REGION Network 61: Step[1301] : JOB[13] Condition
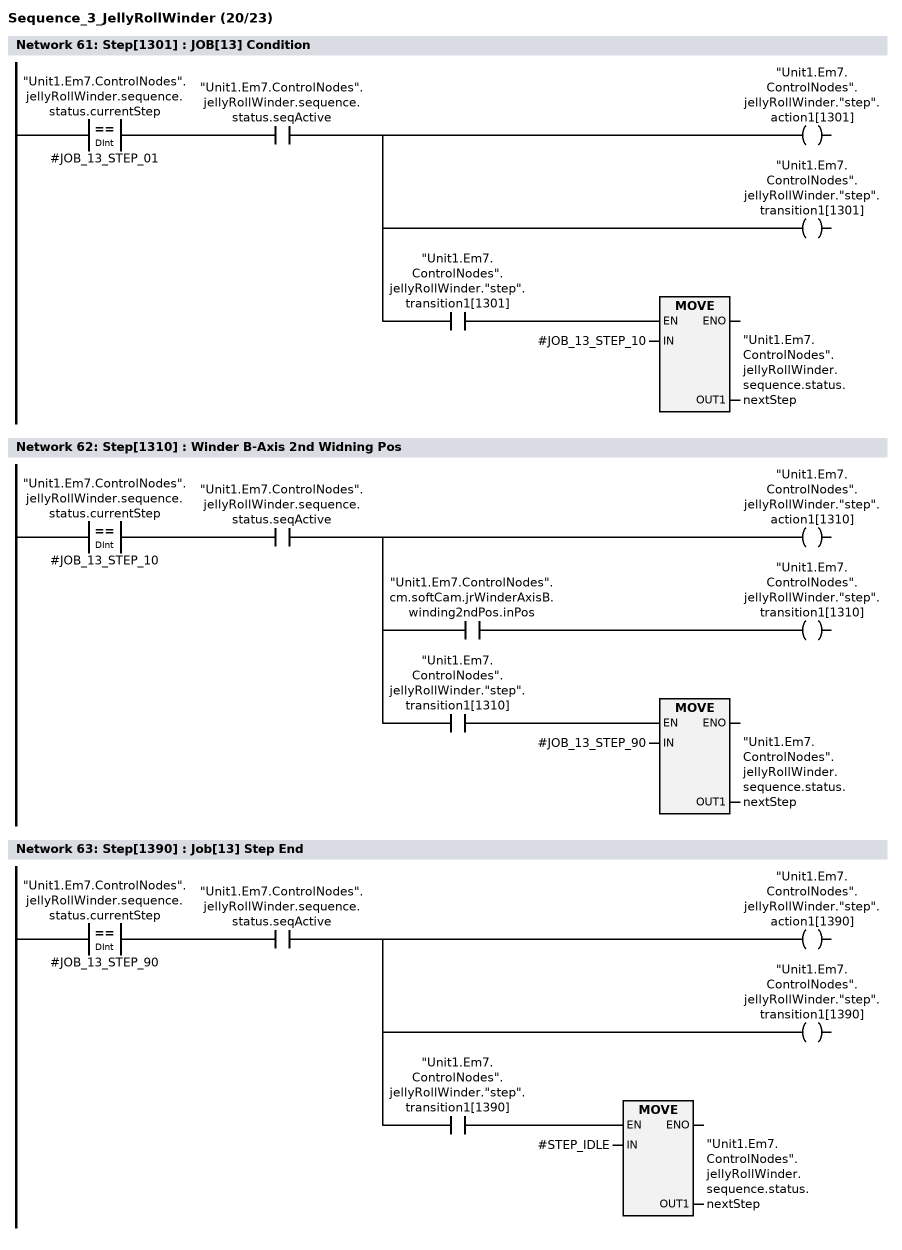
   RUNG wire#powerrail
      { S7_Templates := "SrcType := DInt" } EQ_Contact(in1 := "Unit1.Em7.ControlNodes".jellyRollWinder.sequence.status.currentStep, in2 := #JOB_13_STEP_01)
      Contact( "Unit1.Em7.ControlNodes".jellyRollWinder.sequence.status.seqActive )
      wire#w1
      Coil( "Unit1.Em7.ControlNodes".jellyRollWinder."step".action1[1301] )
   END_RUNG
   RUNG wire#w1
      Coil( "Unit1.Em7.ControlNodes".jellyRollWinder."step".transition1[1301] )
   END_RUNG
   RUNG wire#w1
      Contact( "Unit1.Em7.ControlNodes".jellyRollWinder."step".transition1[1301] )
      Move(in := #JOB_13_STEP_10, out1 => "Unit1.Em7.ControlNodes".jellyRollWinder.sequence.status.nextStep)
   END_RUNG
   // the same network as SCL:
   "Unit1.Em7.ControlNodes".jellyRollWinder."step".action1[1301] := ("Unit1.Em7.ControlNodes".jellyRollWinder.sequence.status.currentStep = #JOB_13_STEP_01) AND "Unit1.Em7.ControlNodes".jellyRollWinder.sequence.status.seqActive;
   "Unit1.Em7.ControlNodes".jellyRollWinder."step".transition1[1301] := ("Unit1.Em7.ControlNodes".jellyRollWinder.sequence.status.currentStep = #JOB_13_STEP_01) AND "Unit1.Em7.ControlNodes".jellyRollWinder.sequence.status.seqActive;
   IF ("Unit1.Em7.ControlNodes".jellyRollWinder.sequence.status.currentStep = #JOB_13_STEP_01) AND "Unit1.Em7.ControlNodes".jellyRollWinder.sequence.status.seqActive AND "Unit1.Em7.ControlNodes".jellyRollWinder."step".transition1[1301] THEN
       "Unit1.Em7.ControlNodes".jellyRollWinder.sequence.status.nextStep := #JOB_13_STEP_10;
   END_IF;
END_REGION

REGION Network 62: Step[1310] : Winder B-Axis 2nd Widning Pos
   RUNG wire#powerrail
      { S7_Templates := "SrcType := DInt" } EQ_Contact(in1 := "Unit1.Em7.ControlNodes".jellyRollWinder.sequence.status.currentStep, in2 := #JOB_13_STEP_10)
      Contact( "Unit1.Em7.ControlNodes".jellyRollWinder.sequence.status.seqActive )
      wire#w1
      Coil( "Unit1.Em7.ControlNodes".jellyRollWinder."step".action1[1310] )
   END_RUNG
   RUNG wire#w1
      Contact( "Unit1.Em7.ControlNodes".cm.softCam.jrWinderAxisB.winding2ndPos.inPos )
      Coil( "Unit1.Em7.ControlNodes".jellyRollWinder."step".transition1[1310] )
   END_RUNG
   RUNG wire#w1
      Contact( "Unit1.Em7.ControlNodes".jellyRollWinder."step".transition1[1310] )
      Move(in := #JOB_13_STEP_90, out1 => "Unit1.Em7.ControlNodes".jellyRollWinder.sequence.status.nextStep)
   END_RUNG
   // the same network as SCL:
   "Unit1.Em7.ControlNodes".jellyRollWinder."step".action1[1310] := ("Unit1.Em7.ControlNodes".jellyRollWinder.sequence.status.currentStep = #JOB_13_STEP_10) AND "Unit1.Em7.ControlNodes".jellyRollWinder.sequence.status.seqActive;
   "Unit1.Em7.ControlNodes".jellyRollWinder."step".transition1[1310] := ("Unit1.Em7.ControlNodes".jellyRollWinder.sequence.status.currentStep = #JOB_13_STEP_10) AND "Unit1.Em7.ControlNodes".jellyRollWinder.sequence.status.seqActive AND "Unit1.Em7.ControlNodes".cm.softCam.jrWinderAxisB.winding2ndPos.inPos;
   IF ("Unit1.Em7.ControlNodes".jellyRollWinder.sequence.status.currentStep = #JOB_13_STEP_10) AND "Unit1.Em7.ControlNodes".jellyRollWinder.sequence.status.seqActive AND "Unit1.Em7.ControlNodes".jellyRollWinder."step".transition1[1310] THEN
       "Unit1.Em7.ControlNodes".jellyRollWinder.sequence.status.nextStep := #JOB_13_STEP_90;
   END_IF;
END_REGION

REGION Network 63: Step[1390] : Job[13] Step End
   RUNG wire#powerrail
      { S7_Templates := "SrcType := DInt" } EQ_Contact(in1 := "Unit1.Em7.ControlNodes".jellyRollWinder.sequence.status.currentStep, in2 := #JOB_13_STEP_90)
      Contact( "Unit1.Em7.ControlNodes".jellyRollWinder.sequence.status.seqActive )
      wire#w1
      Coil( "Unit1.Em7.ControlNodes".jellyRollWinder."step".action1[1390] )
   END_RUNG
   RUNG wire#w1
      Coil( "Unit1.Em7.ControlNodes".jellyRollWinder."step".transition1[1390] )
   END_RUNG
   RUNG wire#w1
      Contact( "Unit1.Em7.ControlNodes".jellyRollWinder."step".transition1[1390] )
      Move(in := #STEP_IDLE, out1 => "Unit1.Em7.ControlNodes".jellyRollWinder.sequence.status.nextStep)
   END_RUNG
   // the same network as SCL:
   "Unit1.Em7.ControlNodes".jellyRollWinder."step".action1[1390] := ("Unit1.Em7.ControlNodes".jellyRollWinder.sequence.status.currentStep = #JOB_13_STEP_90) AND "Unit1.Em7.ControlNodes".jellyRollWinder.sequence.status.seqActive;
   "Unit1.Em7.ControlNodes".jellyRollWinder."step".transition1[1390] := ("Unit1.Em7.ControlNodes".jellyRollWinder.sequence.status.currentStep = #JOB_13_STEP_90) AND "Unit1.Em7.ControlNodes".jellyRollWinder.sequence.status.seqActive;
   IF ("Unit1.Em7.ControlNodes".jellyRollWinder.sequence.status.currentStep = #JOB_13_STEP_90) AND "Unit1.Em7.ControlNodes".jellyRollWinder.sequence.status.seqActive AND "Unit1.Em7.ControlNodes".jellyRollWinder."step".transition1[1390] THEN
       "Unit1.Em7.ControlNodes".jellyRollWinder.sequence.status.nextStep := #STEP_IDLE;
   END_IF;
END_REGION

REGION Network 64: *************** JOB[14] Cam Stop Sync ************************
END_REGION

REGION Network 65: Step[1401] : JOB[14] Condition
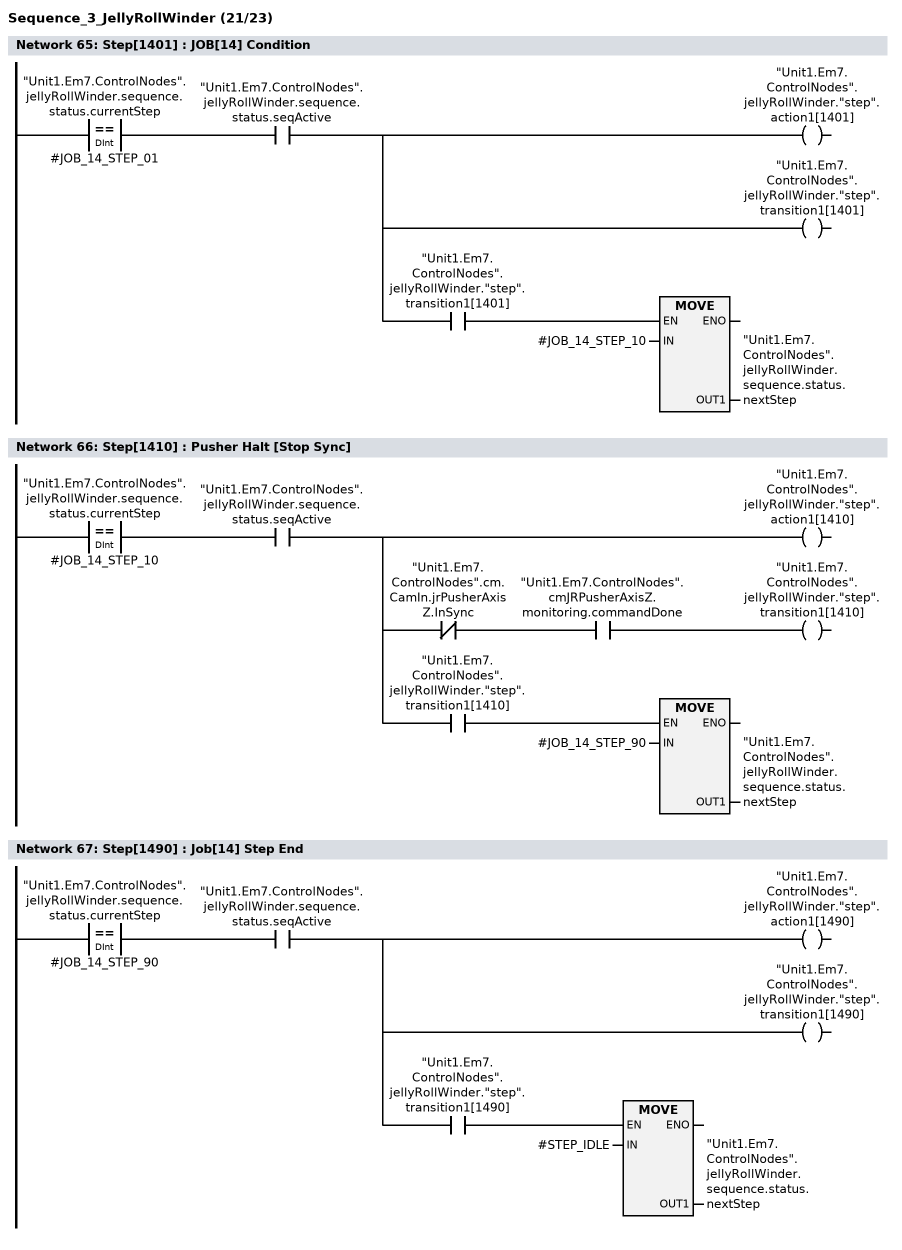
   RUNG wire#powerrail
      { S7_Templates := "SrcType := DInt" } EQ_Contact(in1 := "Unit1.Em7.ControlNodes".jellyRollWinder.sequence.status.currentStep, in2 := #JOB_14_STEP_01)
      Contact( "Unit1.Em7.ControlNodes".jellyRollWinder.sequence.status.seqActive )
      wire#w1
      Coil( "Unit1.Em7.ControlNodes".jellyRollWinder."step".action1[1401] )
   END_RUNG
   RUNG wire#w1
      Coil( "Unit1.Em7.ControlNodes".jellyRollWinder."step".transition1[1401] )
   END_RUNG
   RUNG wire#w1
      Contact( "Unit1.Em7.ControlNodes".jellyRollWinder."step".transition1[1401] )
      Move(in := #JOB_14_STEP_10, out1 => "Unit1.Em7.ControlNodes".jellyRollWinder.sequence.status.nextStep)
   END_RUNG
   // the same network as SCL:
   "Unit1.Em7.ControlNodes".jellyRollWinder."step".action1[1401] := ("Unit1.Em7.ControlNodes".jellyRollWinder.sequence.status.currentStep = #JOB_14_STEP_01) AND "Unit1.Em7.ControlNodes".jellyRollWinder.sequence.status.seqActive;
   "Unit1.Em7.ControlNodes".jellyRollWinder."step".transition1[1401] := ("Unit1.Em7.ControlNodes".jellyRollWinder.sequence.status.currentStep = #JOB_14_STEP_01) AND "Unit1.Em7.ControlNodes".jellyRollWinder.sequence.status.seqActive;
   IF ("Unit1.Em7.ControlNodes".jellyRollWinder.sequence.status.currentStep = #JOB_14_STEP_01) AND "Unit1.Em7.ControlNodes".jellyRollWinder.sequence.status.seqActive AND "Unit1.Em7.ControlNodes".jellyRollWinder."step".transition1[1401] THEN
       "Unit1.Em7.ControlNodes".jellyRollWinder.sequence.status.nextStep := #JOB_14_STEP_10;
   END_IF;
END_REGION

REGION Network 66: Step[1410] : Pusher Halt [Stop Sync]
   RUNG wire#powerrail
      { S7_Templates := "SrcType := DInt" } EQ_Contact(in1 := "Unit1.Em7.ControlNodes".jellyRollWinder.sequence.status.currentStep, in2 := #JOB_14_STEP_10)
      Contact( "Unit1.Em7.ControlNodes".jellyRollWinder.sequence.status.seqActive )
      wire#w1
      Coil( "Unit1.Em7.ControlNodes".jellyRollWinder."step".action1[1410] )
   END_RUNG
   RUNG wire#w1
      I_Contact( "Unit1.Em7.ControlNodes".cm.CamIn.jrPusherAxisZ.InSync )
      Contact( "Unit1.Em7.ControlNodes".cmJRPusherAxisZ.monitoring.commandDone )
      Coil( "Unit1.Em7.ControlNodes".jellyRollWinder."step".transition1[1410] )
   END_RUNG
   RUNG wire#w1
      Contact( "Unit1.Em7.ControlNodes".jellyRollWinder."step".transition1[1410] )
      Move(in := #JOB_14_STEP_90, out1 => "Unit1.Em7.ControlNodes".jellyRollWinder.sequence.status.nextStep)
   END_RUNG
   // the same network as SCL:
   "Unit1.Em7.ControlNodes".jellyRollWinder."step".action1[1410] := ("Unit1.Em7.ControlNodes".jellyRollWinder.sequence.status.currentStep = #JOB_14_STEP_10) AND "Unit1.Em7.ControlNodes".jellyRollWinder.sequence.status.seqActive;
   "Unit1.Em7.ControlNodes".jellyRollWinder."step".transition1[1410] := ("Unit1.Em7.ControlNodes".jellyRollWinder.sequence.status.currentStep = #JOB_14_STEP_10) AND "Unit1.Em7.ControlNodes".jellyRollWinder.sequence.status.seqActive AND NOT "Unit1.Em7.ControlNodes".cm.CamIn.jrPusherAxisZ.InSync AND "Unit1.Em7.ControlNodes".cmJRPusherAxisZ.monitoring.commandDone;
   IF ("Unit1.Em7.ControlNodes".jellyRollWinder.sequence.status.currentStep = #JOB_14_STEP_10) AND "Unit1.Em7.ControlNodes".jellyRollWinder.sequence.status.seqActive AND "Unit1.Em7.ControlNodes".jellyRollWinder."step".transition1[1410] THEN
       "Unit1.Em7.ControlNodes".jellyRollWinder.sequence.status.nextStep := #JOB_14_STEP_90;
   END_IF;
END_REGION

REGION Network 67: Step[1490] : Job[14] Step End
   RUNG wire#powerrail
      { S7_Templates := "SrcType := DInt" } EQ_Contact(in1 := "Unit1.Em7.ControlNodes".jellyRollWinder.sequence.status.currentStep, in2 := #JOB_14_STEP_90)
      Contact( "Unit1.Em7.ControlNodes".jellyRollWinder.sequence.status.seqActive )
      wire#w1
      Coil( "Unit1.Em7.ControlNodes".jellyRollWinder."step".action1[1490] )
   END_RUNG
   RUNG wire#w1
      Coil( "Unit1.Em7.ControlNodes".jellyRollWinder."step".transition1[1490] )
   END_RUNG
   RUNG wire#w1
      Contact( "Unit1.Em7.ControlNodes".jellyRollWinder."step".transition1[1490] )
      Move(in := #STEP_IDLE, out1 => "Unit1.Em7.ControlNodes".jellyRollWinder.sequence.status.nextStep)
   END_RUNG
   // the same network as SCL:
   "Unit1.Em7.ControlNodes".jellyRollWinder."step".action1[1490] := ("Unit1.Em7.ControlNodes".jellyRollWinder.sequence.status.currentStep = #JOB_14_STEP_90) AND "Unit1.Em7.ControlNodes".jellyRollWinder.sequence.status.seqActive;
   "Unit1.Em7.ControlNodes".jellyRollWinder."step".transition1[1490] := ("Unit1.Em7.ControlNodes".jellyRollWinder.sequence.status.currentStep = #JOB_14_STEP_90) AND "Unit1.Em7.ControlNodes".jellyRollWinder.sequence.status.seqActive;
   IF ("Unit1.Em7.ControlNodes".jellyRollWinder.sequence.status.currentStep = #JOB_14_STEP_90) AND "Unit1.Em7.ControlNodes".jellyRollWinder.sequence.status.seqActive AND "Unit1.Em7.ControlNodes".jellyRollWinder."step".transition1[1490] THEN
       "Unit1.Em7.ControlNodes".jellyRollWinder.sequence.status.nextStep := #STEP_IDLE;
   END_IF;
END_REGION

REGION Network 68: *************** IMMEDIATE STOP **************************
END_REGION

REGION Network 69: Immediate Stop
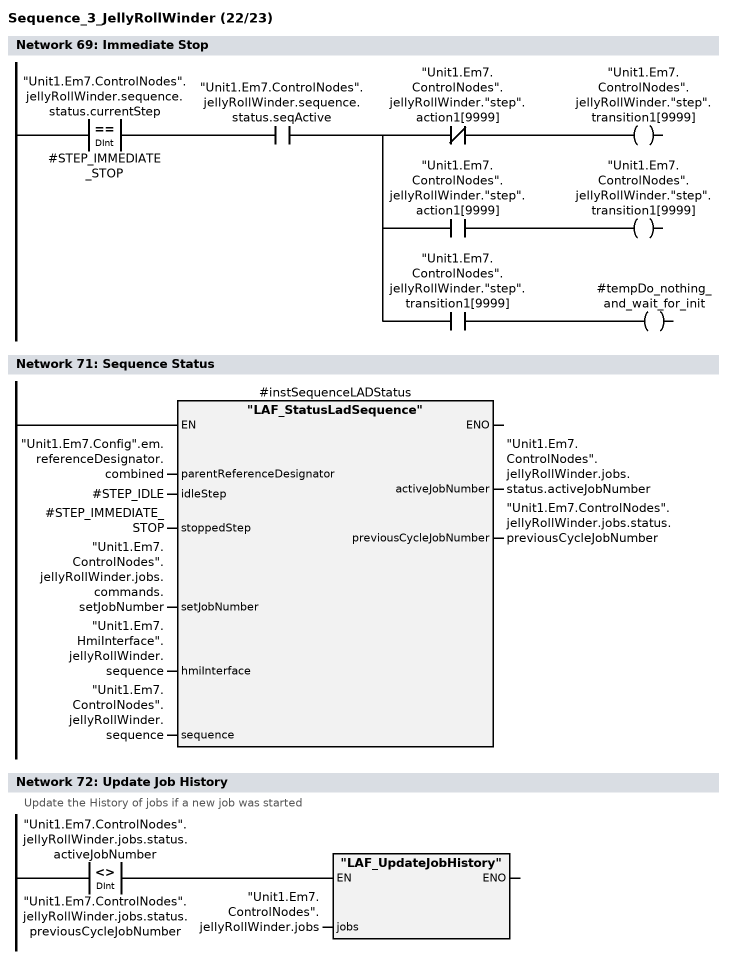
   RUNG wire#powerrail
      { S7_Templates := "SrcType := DInt" } EQ_Contact(in1 := "Unit1.Em7.ControlNodes".jellyRollWinder.sequence.status.currentStep, in2 := #STEP_IMMEDIATE_STOP)
      Contact( "Unit1.Em7.ControlNodes".jellyRollWinder.sequence.status.seqActive )
      wire#w1
      I_Contact( "Unit1.Em7.ControlNodes".jellyRollWinder."step".action1[9999] )
      Coil( "Unit1.Em7.ControlNodes".jellyRollWinder."step".transition1[9999] )
   END_RUNG
   RUNG wire#w1
      Contact( "Unit1.Em7.ControlNodes".jellyRollWinder."step".action1[9999] )
      Coil( "Unit1.Em7.ControlNodes".jellyRollWinder."step".transition1[9999] )
   END_RUNG
   RUNG wire#w1
      Contact( "Unit1.Em7.ControlNodes".jellyRollWinder."step".transition1[9999] )
      Coil( #tempDo_nothing_and_wait_for_init )
   END_RUNG
   // the same network as SCL:
   #_w1 := ("Unit1.Em7.ControlNodes".jellyRollWinder.sequence.status.currentStep = #STEP_IMMEDIATE_STOP) AND "Unit1.Em7.ControlNodes".jellyRollWinder.sequence.status.seqActive;
   "Unit1.Em7.ControlNodes".jellyRollWinder."step".transition1[9999] := #_w1 AND NOT "Unit1.Em7.ControlNodes".jellyRollWinder."step".action1[9999];
   "Unit1.Em7.ControlNodes".jellyRollWinder."step".transition1[9999] := #_w1 AND "Unit1.Em7.ControlNodes".jellyRollWinder."step".action1[9999];
   #tempDo_nothing_and_wait_for_init := #_w1 AND "Unit1.Em7.ControlNodes".jellyRollWinder."step".transition1[9999];
END_REGION

REGION Network 70: *************** Status updates **************************
END_REGION

REGION Network 71: Sequence Status
   RUNG wire#powerrail
      #instSequenceLADStatus(parentReferenceDesignator := "Unit1.Em7.Config".em.referenceDesignator.combined, idleStep := #STEP_IDLE, stoppedStep := #STEP_IMMEDIATE_STOP, setJobNumber := "Unit1.Em7.ControlNodes".jellyRollWinder.jobs.commands.setJobNumber, hmiInterface := "Unit1.Em7.HmiInterface".jellyRollWinder.sequence, sequence := "Unit1.Em7.ControlNodes".jellyRollWinder.sequence, activeJobNumber => "Unit1.Em7.ControlNodes".jellyRollWinder.jobs.status.activeJobNumber, previousCycleJobNumber => "Unit1.Em7.ControlNodes".jellyRollWinder.jobs.status.previousCycleJobNumber)
   END_RUNG
   // the same network as SCL:
   #instSequenceLADStatus(parentReferenceDesignator := "Unit1.Em7.Config".em.referenceDesignator.combined,   // "LAF_StatusLadSequence"
                          idleStep := #STEP_IDLE,
                          stoppedStep := #STEP_IMMEDIATE_STOP,
                          setJobNumber := "Unit1.Em7.ControlNodes".jellyRollWinder.jobs.commands.setJobNumber,
                          hmiInterface := "Unit1.Em7.HmiInterface".jellyRollWinder.sequence,
                          sequence := "Unit1.Em7.ControlNodes".jellyRollWinder.sequence,
                          activeJobNumber => "Unit1.Em7.ControlNodes".jellyRollWinder.jobs.status.activeJobNumber,
                          previousCycleJobNumber => "Unit1.Em7.ControlNodes".jellyRollWinder.jobs.status.previousCycleJobNumber);
END_REGION

REGION Network 72: Update Job History
   // Update the History of jobs if a new job was started
   RUNG wire#powerrail
      { S7_Templates := "SrcType := DInt" } NE_Contact(in1 := "Unit1.Em7.ControlNodes".jellyRollWinder.jobs.status.activeJobNumber, in2 := "Unit1.Em7.ControlNodes".jellyRollWinder.jobs.status.previousCycleJobNumber)
      "LAF_UpdateJobHistory"(jobs := "Unit1.Em7.ControlNodes".jellyRollWinder.jobs)
   END_RUNG
   // the same network as SCL:
   IF "Unit1.Em7.ControlNodes".jellyRollWinder.jobs.status.activeJobNumber <> "Unit1.Em7.ControlNodes".jellyRollWinder.jobs.status.previousCycleJobNumber THEN
       "LAF_UpdateJobHistory"(jobs := "Unit1.Em7.ControlNodes".jellyRollWinder.jobs);
   END_IF;
END_REGION

REGION Network 73: Output steps as String
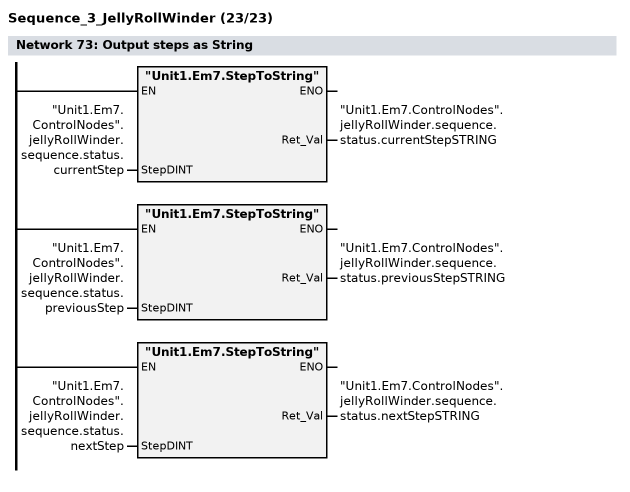
   RUNG wire#powerrail
      "Unit1.Em7.StepToString"(StepDINT := "Unit1.Em7.ControlNodes".jellyRollWinder.sequence.status.currentStep, Ret_Val => "Unit1.Em7.ControlNodes".jellyRollWinder.sequence.status.currentStepSTRING)
   END_RUNG
   RUNG wire#powerrail
      "Unit1.Em7.StepToString"(StepDINT := "Unit1.Em7.ControlNodes".jellyRollWinder.sequence.status.previousStep, Ret_Val => "Unit1.Em7.ControlNodes".jellyRollWinder.sequence.status.previousStepSTRING)
   END_RUNG
   RUNG wire#powerrail
      "Unit1.Em7.StepToString"(StepDINT := "Unit1.Em7.ControlNodes".jellyRollWinder.sequence.status.nextStep, Ret_Val => "Unit1.Em7.ControlNodes".jellyRollWinder.sequence.status.nextStepSTRING)
   END_RUNG
   // the same network as SCL:
   "Unit1.Em7.ControlNodes".jellyRollWinder.sequence.status.currentStepSTRING := "Unit1.Em7.StepToString"(StepDINT := "Unit1.Em7.ControlNodes".jellyRollWinder.sequence.status.currentStep);
   "Unit1.Em7.ControlNodes".jellyRollWinder.sequence.status.previousStepSTRING := "Unit1.Em7.StepToString"(StepDINT := "Unit1.Em7.ControlNodes".jellyRollWinder.sequence.status.previousStep);
   "Unit1.Em7.ControlNodes".jellyRollWinder.sequence.status.nextStepSTRING := "Unit1.Em7.StepToString"(StepDINT := "Unit1.Em7.ControlNodes".jellyRollWinder.sequence.status.nextStep);
END_REGION
END_FUNCTION_BLOCK
